RoboDK station: Decoupe SPUD V2.rdk

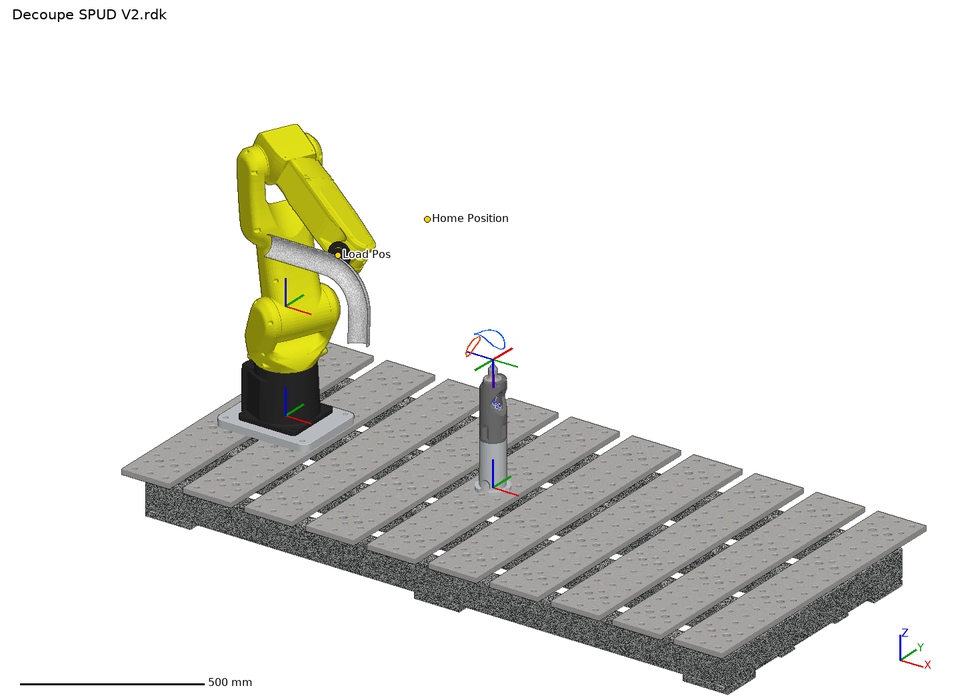
[picture v0: the station drawn from its stored meshes, robots at their saved joint values, targets as dots, program paths as lines]
Station Decoupe SPUD V2 (saved by RoboDK 5.2.1). Poses are relative to the parent item; angles as X-Y-Z fixed-axis rotations.
Station parameters (name, value as stored): IO_5, 1
  - frame LR Mate 200iD/7L Base at (0, 0, 330) mm
    - robot Fanuc LR Mate 200iD/7L: 6 axes, payload 7 kg, reach 911 mm, repeatability 0.03 mm, weight 27 kg
        modified DH rows (alpha deg, a mm, theta deg, d mm): 0, 0, 0, 330; -90, 50, -90, 0; 0, 440, 0, 0; -90, 35, 0, 420; 90, 0, 0, 0; -90, 0, 0, 80
        base shift (0, 0, -330) mm
        joint limits [-170, -70, -70, -190, -115, -360] to [170, 145, 215, 190, 115, 360]; home [0, 0, 0, 0, 0, 0]; saved at [-25.048, -11.03, -19.278, 110.835, -71.299, -25.474]
      - tool ZIPPER - 2201 - COQUILLE, TCP at (0, 0, 0) mm, size 365.9 x 230.6 x 35 mm, geometry from ZIPPER - 2200 - ASSEMBLAGE SUPPORT COQUILLE.step
      - tool COUPE 2, TCP at (0, 0, 0) mm
      - tool COUPE 1, TCP at (0, 0, 0) mm
    - frame ORIGINE TABLE at (0, 0, -330) mm
      - object ZIPPER - 5100 - TABLE ROBOT at (0, 0, 0) mm, size 1988.8 x 965.2 x 186.4 mm, geometry from coquille.step
      - frame ORIGINE COUTEAU at (685.8, 0, -25.4) mm
        - frame TCP LAME 2 at (0, 0, 387.45) mm, rotated rx 0 ry 90 rz 180 deg
        - frame TCP LAME 1 at (0, 0, 387.45) mm, rotated rx 178.24 ry -0.1 rz 86.85 deg
        - object ZIPPER - 3200 - ASSEMBLAGE DECOUPE 3D at (0, 0, 0) mm, size 98.8 x 97.7 x 387.5 mm, geometry from ZIPPER - 3200 - ASSEMBLAGE DECOUPE 3D.step
    - target Home Position (joint target) at (470, 0, 395) mm, rotated rx -180 ry 0 rz 0 deg; joints [0, 0, 0, 0, -90, 0] of Fanuc LR Mate 200iD/7L
    - target Load Pos (Cartesian target) at (338.68, -236.45, 343.22) mm, rotated rx 77.75 ry 0 rz 0.01 deg; joints [-25.048, -11.03, -19.278, 110.835, -71.299, -25.474] of Fanuc LR Mate 200iD/7L
  - machining project TOURSPUD 1: onStart | onPathStart | onApproach | onPoint | onRetract | onFinish | SetRPM(%1) | SetTool(%1) | Extruder(%1) | default | default | OutOnMov(%1) | OutOffMov(%1) | onPathFinish | M_RunCode(%1)
  - machining project TOURSPUD 2: onStart | onPathStart | onApproach | onPoint | onRetract | onFinish | SetRPM(%1) | SetTool(%1) | Extruder(%1) | default | default | OutOnMov(%1) | OutOffMov(%1) | onPathFinish | M_RunCode(%1)
  - program TOURSPUD 2 (43 instructions, listed below)
  - program TOURSPUD 1 (43 instructions, listed below)
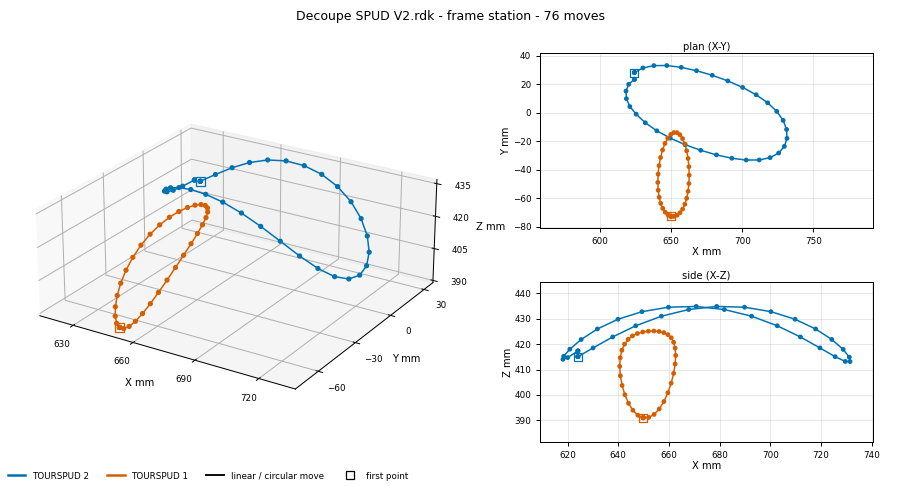
[picture p0: tool path of Decoupe SPUD V2.rdk in frame station, 76 of 76 moves have a stored position in this frame; points joined in program order, loops and branches not executed]

--- program TOURSPUD 2 (robot Fanuc LR Mate 200iD/7L) ---
  Smooth(1)
  Set Ref.: TCP LAME 2
  Set Tool: ZIPPER - 2201 - COQUILLE
  Show ZIPPER - 2201 - COQUILLE
  MoveJ 1 to (-53.02, -28.3, 61.73) mm, rotated rx -120 ry -5.27 rz -86.96 deg; joints [2.773, 25.601, -39.866, 3.972, -20.347, 89.95]
  MoveL 2 to (-53.02, -28.3, 61.73) mm, rotated rx -120 ry -5.27 rz -86.96 deg; joints [2.773, 25.601, -39.866, 3.972, -20.347, 89.95]
  MoveL 3 to (-53.02, -28.3, 61.73) mm, rotated rx -120 ry -5.27 rz -86.96 deg; joints [2.773, 25.601, -39.866, 3.972, -20.347, 89.95]
  MoveL 4 to (-53.02, -28.3, 61.73) mm, rotated rx -120 ry -5.27 rz -86.96 deg; joints [2.773, 25.601, -39.866, 3.972, -20.347, 89.95]
  Set speed (10.0 mm/s)
  MoveL 5 to (-56.46, -31.54, 55.74) mm, rotated rx -120 ry 6.06 rz -93.49 deg; joints [3.059, 26.012, -39.065, 4.206, -21.207, 76.433]
  MoveL 6 to (-60.8, -33.17, 48) mm, rotated rx -120 ry 17.4 rz -99.8 deg; joints [3.166, 26.66, -37.848, 3.754, -23.736, 63.886]
  MoveL 7 to (-65.2, -33.23, 38.92) mm, rotated rx -120 ry 28.62 rz -105.46 deg; joints [3.109, 27.581, -36.368, 2.94, -27.661, 52.389]
  MoveL 8 to (-68.98, -31.95, 28.79) mm, rotated rx -120 ry 39.82 rz -110.29 deg; joints [2.921, 28.813, -34.749, 2.075, -32.712, 41.643]
  MoveL 9 to (-71.61, -29.6, 18.01) mm, rotated rx -120 ry 50.99 rz -114.16 deg; joints [2.637, 30.355, -33.106, 1.331, -38.575, 31.508]
  MoveL 10 to (-72.83, -26.38, 6.98) mm, rotated rx -120 ry 62.15 rz -117.04 deg; joints [2.288, 32.18, -31.52, 0.756, -44.987, 21.824]
  MoveL 11 to (-72.52, -22.42, -4.02) mm, rotated rx -120 ry 73.43 rz -118.96 deg; joints [1.893, 34.254, -30.035, 0.343, -51.772, 12.362]
  MoveL 12 to (-70.77, -17.84, -14.42) mm, rotated rx -120 ry 84.7 rz -119.89 deg; joints [1.468, 36.477, -28.711, 0.079, -58.642, 3.086]
  MoveL 13 to (-67.77, -12.67, -23.93) mm, rotated rx 60 ry 83.93 rz 60.14 deg; joints [1.017, 38.773, -27.565, -0.059, -65.466, -6.253]
  MoveL 14 to (-63.95, -7.03, -32.02) mm, rotated rx 60 ry 72.63 rz 61.14 deg; joints [0.552, 40.999, -26.631, -0.087, -71.955, -15.68]
  MoveL 15 to (-59.8, -0.99, -38.41) mm, rotated rx 60 ry 61.37 rz 63.13 deg; joints [0.076, 43.041, -25.913, -0.019, -77.948, -25.371]
  MoveL 16 to (-55.88, 5.34, -42.9) mm, rotated rx 60 ry 50.15 rz 66.09 deg; joints [-0.406, 44.784, -25.406, 0.131, -83.278, -35.488]
  MoveL 17 to (-52.82, 11.72, -45.32) mm, rotated rx 60 ry 39.02 rz 70.02 deg; joints [-0.881, 46.11, -25.099, 0.343, -87.757, -46.101]
  MoveL 18 to (-51.09, 17.96, -45.61) mm, rotated rx 60 ry 27.82 rz 74.92 deg; joints [-1.342, 46.937, -24.965, 0.594, -91.275, -57.434]
  MoveL 19 to (-51.13, 23.62, -43.74) mm, rotated rx 60 ry 16.6 rz 80.64 deg; joints [-1.762, 47.182, -24.983, 0.846, -93.637, -69.408]
  MoveL 20 to (-53.01, 28.29, -39.73) mm, rotated rx 60 ry 5.28 rz 86.96 deg; joints [-2.117, 46.808, -25.135, 1.057, -94.707, -81.981]
  MoveL 21 to (-56.46, 31.54, -33.73) mm, rotated rx 60 ry -6.07 rz 93.49 deg; joints [-2.379, 45.829, -25.419, 1.186, -94.373, -94.846]
  MoveL 22 to (-60.79, 33.17, -26.03) mm, rotated rx 60 ry -17.36 rz 99.77 deg; joints [-2.532, 44.334, -25.843, 1.209, -92.637, -107.566]
  MoveL 23 to (-65.21, 33.23, -16.91) mm, rotated rx 60 ry -28.64 rz 105.47 deg; joints [-2.579, 42.433, -26.431, 1.131, -89.577, -119.922]
  MoveL 24 to (-68.98, 31.96, -6.79) mm, rotated rx 60 ry -39.82 rz 110.29 deg; joints [-2.53, 40.276, -27.193, 0.974, -85.373, -131.651]
  MoveL 25 to (-71.61, 29.6, 3.97) mm, rotated rx 60 ry -50.97 rz 114.16 deg; joints [-2.397, 37.981, -28.14, 0.766, -80.196, -142.789]
  MoveL 26 to (-72.83, 26.37, 15.06) mm, rotated rx 60 ry -62.19 rz 117.05 deg; joints [-2.19, 35.65, -29.278, 0.531, -74.203, -153.463]
  MoveL 27 to (-72.53, 22.43, 25.99) mm, rotated rx 60 ry -73.4 rz 118.96 deg; joints [-1.914, 33.404, -30.584, 0.296, -67.625, -163.742]
  MoveL 28 to (-70.76, 17.82, 36.46) mm, rotated rx 60 ry -84.75 rz 119.9 deg; joints [-1.564, 31.312, -32.047, 0.082, -60.576, -173.927]
  MoveL 29 to (-67.77, 12.68, 45.92) mm, rotated rx -120 ry -83.94 rz -60.14 deg; joints [-1.143, 29.49, -33.601, -0.075, -53.375, -184.065]
  MoveL 30 to (-63.94, 7.02, 54.03) mm, rotated rx -120 ry -72.61 rz -61.15 deg; joints [-0.649, 27.983, -35.194, -0.134, -46.211, -194.443]
  MoveL 31 to (-59.78, 0.97, 60.43) mm, rotated rx -120 ry -61.33 rz -63.13 deg; joints [-0.091, 26.835, -36.729, -0.034, -39.393, -205.223]
  MoveL 32 to (-55.97, -4.36, 64.9) mm, rotated rx -120 ry -50.16 rz -67.09 deg; joints [0.292, 26.037, -38.09, -1.558, -33.23, -215.144]
  MoveL 33 to (-53.18, -9.91, 67.32) mm, rotated rx -120 ry -38.97 rz -72.04 deg; joints [0.715, 25.537, -39.166, -3.337, -27.966, -225.444]
  MoveL 34 to (-51.96, -15.27, 67.61) mm, rotated rx -120 ry -27.81 rz -77.92 deg; joints [1.132, 25.292, -39.833, -5.401, -23.939, -236.06]
  MoveL 35 to (-52.65, -20.02, 65.73) mm, rotated rx -120 ry -16.56 rz -84.66 deg; joints [1.489, 25.254, -40.007, -7.678, -21.4, -247.122]
  MoveL 36 to (-55.28, -23.57, 61.73) mm, rotated rx -120 ry -5.27 rz -91.96 deg; joints [1.718, 25.404, -39.643, -9.93, -20.584, -258.598]
  MoveL 37 to (-55.28, -23.57, 61.73) mm, rotated rx -120 ry -5.27 rz -91.96 deg; joints [1.718, 25.404, -39.643, -9.93, -20.584, -258.598]
  MoveL 38 to (-55.28, -23.57, 61.73) mm, rotated rx -120 ry -5.27 rz -91.96 deg; joints [1.718, 25.404, -39.643, -9.93, -20.584, -258.598]

--- program TOURSPUD 1 (robot Fanuc LR Mate 200iD/7L) ---
  Smooth(1)
  Set Ref.: TCP LAME 1
  Set Tool: ZIPPER - 2201 - COQUILLE
  Show ZIPPER - 2201 - COQUILLE
  MoveJ 1 to (-74.55, -31.01, -30.04) mm, rotated rx -50.69 ry 0 rz -90 deg; joints [-11.785, 36.724, -39.663, -54.503, -70.819, -141.689]
  MoveL 2 to (-74.55, -31.01, -30.04) mm, rotated rx -50.69 ry 0 rz -90 deg; joints [-11.785, 36.724, -39.663, -54.503, -70.819, -141.689]
  MoveL 3 to (-74.55, -31.01, -30.04) mm, rotated rx -50.69 ry 0 rz -90 deg; joints [-11.785, 36.724, -39.663, -54.503, -70.819, -141.689]
  MoveL 4 to (-74.55, -31.01, -30.04) mm, rotated rx -50.69 ry 0 rz -90 deg; joints [-11.785, 36.724, -39.663, -54.503, -70.819, -141.689]
  Set speed (10.0 mm/s)
  MoveL 5 to (-74.52, -28.84, -30.08) mm, rotated rx -50.66 ry 0 rz -90 deg; joints [-11.752, 36.942, -39.474, -54.441, -70.89, -141.876]
  MoveL 6 to (-73.58, -26.71, -31.2) mm, rotated rx -49.79 ry 0 rz -90 deg; joints [-11.579, 36.977, -39.096, -53.687, -70.47, -142.524]
  MoveL 7 to (-71.77, -24.73, -33.28) mm, rotated rx -48.15 ry 0 rz -90 deg; joints [-11.272, 36.841, -38.563, -52.276, -69.613, -143.607]
  MoveL 8 to (-69.09, -22.96, -36.15) mm, rotated rx -45.81 ry 0 rz -90 deg; joints [-10.835, 36.559, -37.907, -50.236, -68.395, -145.113]
  MoveL 9 to (-65.6, -21.45, -39.57) mm, rotated rx -42.91 ry 0 rz -90 deg; joints [-10.275, 36.166, -37.177, -47.621, -66.917, -147.016]
  MoveL 10 to (-61.34, -20.27, -43.3) mm, rotated rx -39.54 ry 0 rz -90 deg; joints [-9.6, 35.694, -36.415, -44.489, -65.279, -149.295]
  MoveL 11 to (-56.37, -19.46, -47.14) mm, rotated rx -35.81 ry 0 rz -90 deg; joints [-8.817, 35.176, -35.66, -40.875, -63.573, -151.936]
  MoveL 12 to (-50.88, -19.05, -50.82) mm, rotated rx -31.88 ry 0 rz -90 deg; joints [-7.955, 34.647, -34.96, -36.913, -61.915, -154.859]
  MoveL 13 to (-45.01, -19.06, -54.19) mm, rotated rx -27.85 ry 0 rz -90 deg; joints [-7.032, 34.129, -34.342, -32.683, -60.377, -158.01]
  MoveL 14 to (-39.06, -19.5, -57.08) mm, rotated rx -23.92 ry 0 rz -90 deg; joints [-6.096, 33.648, -33.838, -28.399, -59.047, -161.233]
  MoveL 15 to (-33.29, -20.34, -59.42) mm, rotated rx -20.21 ry 0 rz -90 deg; joints [-5.186, 33.215, -33.46, -24.231, -57.955, -164.398]
  MoveL 16 to (-27.94, -21.55, -61.21) mm, rotated rx -16.86 ry 0 rz -90 deg; joints [-4.34, 32.829, -33.205, -20.363, -57.104, -167.358]
  MoveL 17 to (-23.31, -23.07, -62.49) mm, rotated rx -14 ry 0 rz -90 deg; joints [-3.604, 32.489, -33.066, -17.001, -56.475, -169.946]
  MoveL 18 to (-19.55, -24.87, -63.34) mm, rotated rx -11.71 ry 0 rz -90 deg; joints [-3.005, 32.181, -33.026, -14.279, -56.02, -172.051]
  MoveL 19 to (-16.93, -26.86, -63.85) mm, rotated rx -10.12 ry 0 rz -90 deg; joints [-2.584, 31.899, -33.069, -12.377, -55.697, -173.524]
  MoveL 20 to (-15.59, -28.99, -64.08) mm, rotated rx -9.31 ry 0 rz -90 deg; joints [-2.366, 31.634, -33.179, -11.412, -55.465, -174.266]
  MoveL 21 to (-15.63, -31.16, -64.07) mm, rotated rx -9.34 ry 0 rz -90 deg; joints [-2.371, 31.39, -33.343, -11.47, -55.308, -174.201]
  MoveL 22 to (-17.07, -33.28, -63.83) mm, rotated rx -10.2 ry 0 rz -90 deg; joints [-2.601, 31.178, -33.555, -12.551, -55.235, -173.323]
  MoveL 23 to (-19.79, -35.27, -63.3) mm, rotated rx -11.85 ry 0 rz -90 deg; joints [-3.042, 31.017, -33.816, -14.587, -55.283, -171.679]
  MoveL 24 to (-23.61, -37.04, -62.41) mm, rotated rx -14.18 ry 0 rz -90 deg; joints [-3.663, 30.931, -34.13, -17.434, -55.506, -169.386]
  MoveL 25 to (-28.31, -38.55, -61.1) mm, rotated rx -17.09 ry 0 rz -90 deg; joints [-4.432, 30.943, -34.509, -20.933, -55.963, -166.572]
  MoveL 26 to (-33.7, -39.73, -59.27) mm, rotated rx -20.47 ry 0 rz -90 deg; joints [-5.314, 31.076, -34.96, -24.917, -56.706, -163.383]
  MoveL 27 to (-39.47, -40.54, -56.9) mm, rotated rx -24.18 ry 0 rz -90 deg; joints [-6.259, 31.344, -35.483, -29.158, -57.758, -160.013]
  MoveL 28 to (-45.44, -40.95, -53.96) mm, rotated rx -28.14 ry 0 rz -90 deg; joints [-7.234, 31.755, -36.077, -33.508, -59.126, -156.597]
  MoveL 29 to (-51.27, -40.94, -50.58) mm, rotated rx -32.15 ry 0 rz -90 deg; joints [-8.18, 32.296, -36.716, -37.717, -60.745, -153.348]
  MoveL 30 to (-56.75, -40.5, -46.86) mm, rotated rx -36.09 ry 0 rz -90 deg; joints [-9.064, 32.946, -37.378, -41.657, -62.548, -150.373]
  MoveL 31 to (-61.68, -39.65, -43.02) mm, rotated rx -39.8 ry 0 rz -90 deg; joints [-9.847, 33.666, -38.022, -45.183, -64.415, -147.784]
  MoveL 32 to (-65.88, -38.45, -39.31) mm, rotated rx -43.14 ry 0 rz -90 deg; joints [-10.507, 34.408, -38.607, -48.204, -66.223, -145.642]
  MoveL 33 to (-69.33, -36.92, -35.91) mm, rotated rx -46.01 ry 0 rz -90 deg; joints [-11.037, 35.132, -39.099, -50.695, -67.874, -143.949]
  MoveL 34 to (-71.93, -35.13, -33.11) mm, rotated rx -48.29 ry 0 rz -90 deg; joints [-11.426, 35.786, -39.458, -52.595, -69.248, -142.728]
  MoveL 35 to (-73.68, -33.14, -31.08) mm, rotated rx -49.88 ry 0 rz -90 deg; joints [-11.677, 36.33, -39.655, -53.88, -70.257, -141.972]
  MoveL 36 to (-74.55, -31.01, -30.04) mm, rotated rx -50.69 ry 0 rz -90 deg; joints [-11.785, 36.724, -39.663, -54.503, -70.819, -141.689]
  MoveL 37 to (-74.55, -31.01, -30.04) mm, rotated rx -50.69 ry 0 rz -90 deg; joints [-11.785, 36.724, -39.663, -54.503, -70.819, -141.689]
  MoveL 38 to (-74.55, -31.01, -30.04) mm, rotated rx -50.69 ry 0 rz -90 deg; joints [-11.785, 36.724, -39.663, -54.503, -70.819, -141.689]
